(* PLC project v0.6.04_CycleSemiAuto.project, CODESYS CODESYS V3.5 SP19 Patch 1 *)
(* stored: creationDateTime 2026-08-01T00:07:15.199610, modificationDateTime 2026-08-01T00:07:15.199610 *)

(* ═══════════════════════════════════════════════════════════════ 🔧 ST_BypassBucket — Bypass de la surveillance benne (M2) 🔒 Doctrine : actionnable UNIQUEMENT en MAINT_N2, RETAIN, jamais masque les autres défauts du même bloc. ═══════════════════════════════════════════════════════════════ *)
TYPE ST_BypassBucket : STRUCT
  Global : BOOL;  (* 🛡️ 1. Hiérarchie & Restauration 🌐 Bypass Global : ignore toute surveillance du mécanisme benne *)
  Initialized : BOOL := FALSE;  (* 🐛 FIX persistance (voir DOC/AUDITS/ConfigPersistence/) : flag restauration boot dédié (défaut FALSE non ambigu, contrairement à une valeur métier) — PRG_SUPERVISION_CFC.st 🚦 TRUE = bypass restauré depuis GVL_BypassRetain ce boot *)
END_STRUCT;
END_TYPE
